// TIA Portal V20 export
// export: Created 2026-04-28T10:07:59.704243Z, ExportSetting WithDefaults, DisplayName Totally Integrated Automation Portal, DisplayVersion V20, DisplayName TIA Portal Openness, DisplayVersion V20, DisplayName TIA Portal Version Control Interface, DisplayVersion V20, DisplayName SINAMICS Startdrive Advanced, DisplayVersion V20, DisplayName SINAMICS Startdrive G130, G150, S120, S150, SINAMICS MV, G220, S200, S210, DisplayVersion V20, DisplayName SINAMICS Startdrive G110M, G120, G120C, G120D, G120P, G115D, DisplayVersion V20, DisplayName STEP 7 Professional, DisplayVersion V20, DisplayName STEP 7 Safety, DisplayVersion V20, DisplayName WinCC Basic/Comfort/Advanced, DisplayVersion V20, DisplayName WinCC Unified, DisplayVersion V20
TYPE "Daten_SPT_60"
// stored: IsFailsafeCompliant false
   STRUCT
      xSlPu : Bool := false;   // Selection Slip Pump
      txt_cSlPu_1_2 : DInt := 0;   // Selection Slip Pump 1 or 2
      xSlPuSoll : Bool := false;   // Selection Slip Pump Set Value
      xSlPuIst : Bool := false;   // Selection Slip Pump Actual Value
      txt_rSlPu : DInt := 0;   // Set value Slip pump
      RangeSlPu : DInt := 0;   // Range Slip pump
      iTakt_1_SlPu : DInt := 0;   // Interval for recording the measured values
      iAnzWerte_1_SlP : DInt := 0;   // Number of measured values
      xs1PuIst_Mod : Bool := false;   // Selection 0-20mA = 0 ; 0-10V = 1
      xSlPuSoll2 : Bool := false;   // Selection Slip Pump 2 Set Value
      xSlPuIst2 : Bool := false;   // Selection Slip Pump 2 Actual Value
      txt_rSlPu2 : DInt := 0;   // Set value Slip pump 2
      RangeSlPu2 : DInt := 0;   // Range Slip pump 2
      iTakt_2_SlPu : DInt := 0;   // Interval for recording the measured values
      iAnzWerte_2_SlP : DInt := 0;   // Number of measured values
      xSlip : Bool := false;   // Selection Slip
      xPrSlContr : Bool := false;   // Selection Slip pressure control
      txt_PrSlControll : DInt := 0;   // Slip pressure (control)
      txt_PrSlToleranze : DInt := 0;   // Slip pressure (tolerance)
      txt_iPrSlTime : Time := T#0MS;   // Slip pressure Delay time
      xPrSl : Bool := false;   // Selection Slip pressure
      txt_rPrSlMa : DInt := 0;   // Slip pressure Max
      txt_max_rPrSlMa : DInt := 0;   // Slip pressure Input Limit
      RangeSlPr : DInt := 0;   // Range Slip pressure
      iTakt_PrSl : DInt := 0;   // Interval for recording the measured values
      iAnzWerte_PrSl : DInt := 0;   // Number of measured values
      xPrSl2 : Bool := false;   // Selection Slip pressure 2
      txt_rPrSlMa2 : DInt := 0;   // Slip pressure 2 Max
      txt_max_rPrSlMa2 : DInt := 0;   // Slip pressure 2 Input Limit
      RangeSlPr2 : DInt := 0;   // Range Slip pressure 2
      iTakt_PrSl2 : DInt := 0;   // Interval for recording the measured values
      iAnzWerte_PrSl2 : DInt := 0;   // Number of measured values
      rDiffSl1Sl2_Set : DInt := 0;   // Difference value of slip pressure 1 and 2
      xFlRa : Bool := false;   // Selection Mass flow
      txt_rFlRaMa : DInt := 0;   // Mass flow Max.
      txt_max_rFlRaMa : DInt := 0;   // Mass flow Input Limit
      RangeFlRa : DInt := 0;   // Range Mass flow
      iTakt_FlRa : DInt := 0;   // Interval for recording the measured values
      iAnzWerte_FlRa : DInt := 0;   // Number of measured values
      xMemBreak : Bool := false;   // Selection Membrane break
      xAir : Bool := false;   // Selection Air
      xPrAi : Bool := false;   // Selection Pressure atomizing air
      RangePrAi : DInt := 0;   // Range Pressure atomizing air
      iTakt_PrAi : DInt := 0;   // Interval for recording the measured values
      iAnzWerte_PrAi : DInt := 0;   // Number of measured values
      xCoAi : Bool := false;   // Selection Air flow nozzle
      txt_rCoAiMi : DInt := 0;   // Air flow nozzle Max.
      txt_max_rCoAiMi : DInt := 0;   // Air flow nozzle Input Limit
      RangeCoAi : DInt := 0;   // Range Air flow nozzle
      iTakt_CoAi : DInt := 0;   // Interval for recording the measured values
      iAnzWerte_CoAi : DInt := 0;   // Number of measured values
      xSlSupp : Bool := false;   // Selection Slip feed
      xTankLevel : Bool := false;   // Selection Tank Level
      txt_iTankLevOver : DInt := 0;   // Tank Level Overflow
      txt_iTankLevMax : DInt := 0;   // Tank Level Max.
      txt_iTankLevMin : DInt := 0;   // Tank Level Min.
      iRangeTankLevel : DInt := 0;   // Range Tank Level
      iTakt_TankLevel : DInt := 0;   // Interval for recording the measured values
      iAnW_TankLevel : DInt := 0;   // Number of measured values
      xAgit_1 : Bool := false;   // Selection Agitator 1
      xAgitSoll_1 : Bool := false;   // Selection Agitator 1 Set Value
      xAgitIst_1 : Bool := false;   // Selection Agitator 1 Actual Value
      xAgitSpCon_1 : Bool := false;   // Selection Agitator 1 Speed ​​manual
      iRangeAgit_1 : DInt := 0;   // Range Agitator 1
      iAgitSoll_1 : DInt := 0;   // Set Value Agitator 1
      iTakt_Agit_1 : DInt := 0;   // Interval for recording the measured values
      iAnW_Agit_1 : DInt := 0;   // Number of measured values
      xScAgit_1 : Bool := false;   // Selection Scale agitator 1
      xScAgitSoll_1 : Bool := false;   // Selection Scale agitator 1 Set Value
      xScAgitIst_1 : Bool := false;   // Selection Scale agitator 1 Actual Value
      iRangeScAgit_1 : DInt := 0;   // Range Scale agitator 1
      iScAgitSoll_1 : DInt := 0;   // Set Value Scale agitator 1
      iScAgitMax_1 : DInt := 0;   // Scale agitator 1 Max
      iScAgitMin_1 : DInt := 0;   // Scale agitator 1 Min.
      iScAgitOver_1 : DInt := 0;   // Scale agitator 1 Over
      iTakt_ScAgit_1 : DInt := 0;   // Interval for recording the measured values
      iAnW_ScAgit_1 : DInt := 0;   // Number of measured values
      xAgit_2 : Bool := false;   // Selection Agitator 2
      xAgitSoll_2 : Bool := false;   // Selection Agitator 2 Set Value
      xAgitIst_2 : Bool := false;   // Selection Agitator 2 Actual Value
      xAgitSpCon_2 : Bool := false;   // Selection Agitator 2 Speed ​​manual
      iRangeAgit_2 : DInt := 0;   // Range Agitator 2
      iAgitSoll_2 : DInt := 0;   // Set Value Agitator 2
      iTakt_Agit_2 : DInt := 0;   // Interval for recording the measured values
      iAnW_Agit_2 : DInt := 0;   // Number of measured values
      xScAgit_2 : Bool := false;   // Selection Scale agitator 2
      xScAgitSoll_2 : Bool := false;   // Selection Scale agitator 2 Set Value
      xScAgitIst_2 : Bool := false;   // Selection Scale agitator 2 Actual Value
      iRangeScAgit_2 : DInt := 0;   // Range Scale agitator 2
      iScAgitSoll_2 : DInt := 0;   // Set Value Scale agitator 2
      iScAgitMax_2 : DInt := 0;   // Scale agitator 2 Max
      iScAgitMin_2 : DInt := 0;   // Scale agitator 2 Min.
      iScAgitOver_2 : DInt := 0;   // Scale agitator 2 Over
      iTakt_ScAgit_2 : DInt := 0;   // Interval for recording the measured values
      iAnW_ScAgit_2 : DInt := 0;   // Number of measured values
      xAgit_3 : Bool := false;   // Selection Agitator 3
      xAgitSoll_3 : Bool := false;   // Selection Agitator 3 Set Value
      xAgitIst_3 : Bool := false;   // Selection Agitator 3 Actual Value
      xAgitSpCon_3 : Bool := false;   // Selection Agitator 3 Speed ​​manual
      iRangeAgit_3 : DInt := 0;   // Range Agitator 3
      iAgitSoll_3 : DInt := 0;   // Set Value Agitator 3
      iTakt_Agit_3 : DInt := 0;   // Interval for recording the measured values
      iAnW_Agit_3 : DInt := 0;   // Number of measured values
      xScAgit_3 : Bool := false;   // Selection Scale agitator 3
      xScAgitSoll_3 : Bool := false;   // Selection Scale agitator 3 Set Value
      xScAgitIst_3 : Bool := false;   // Selection Scale agitator 3 Actual Value
      iRangeScAgit_3 : DInt := 0;   // Range Scale agitator 3
      iScAgitSoll_3 : DInt := 0;   // Set Value Scale agitator 3
      iScAgitMax_3 : DInt := 0;   // Scale agitator 3 Max
      iScAgitMin_3 : DInt := 0;   // Scale agitator 3 Min.
      iScAgitOver_3 : DInt := 0;   // Scale agitator 3 Over
      iTakt_ScAgit_3 : DInt := 0;   // Interval for recording the measured values
      iAnW_ScAgit_3 : DInt := 0;   // Number of measured values
      xAgit_4 : Bool := false;   // Selection Agitator 4
      xAgitSoll_4 : Bool := false;   // Selection Agitator 4 Set Value
      xAgitIst_4 : Bool := false;   // Selection Agitator 4 Actual Value
      xAgitSpCon_4 : Bool := false;   // Selection Agitator 4 Speed ​​manual
      iRangeAgit_4 : DInt := 0;   // Range Agitator 4
      iAgitSoll_4 : DInt := 0;   // Set Value Agitator 4
      iTakt_Agit_4 : DInt := 0;   // Interval for recording the measured values
      iAnW_Agit_4 : DInt := 0;   // Number of measured values
      xScAgit_4 : Bool := false;   // Selection Scale agitator 4
      xScAgitSoll_4 : Bool := false;   // Selection Scale agitator 4 Set Value
      xScAgitIst_4 : Bool := false;   // Selection Scale agitator 4 Actual Value
      iRangeScAgit_4 : DInt := 0;   // Range Scale agitator 4
      iScAgitSoll_4 : DInt := 0;   // Set Value Scale agitator 4
      iScAgitMax_4 : DInt := 0;   // Scale agitator 4 Max
      iScAgitMin_4 : DInt := 0;   // Scale agitator 4 Min.
      iScAgitOver_4 : DInt := 0;   // Scale agitator 4 Over
      iTakt_ScAgit_4 : DInt := 0;   // Interval for recording the measured values
      iAnW_ScAgit_4 : DInt := 0;   // Number of measured values
      xOelTemp : Bool := false;   // Selection Oil temperature slip pump
      iRangeOelTemp : DInt := 0;   // Range Oil temperature slip pump
      iTakt_OelTemp : DInt := 0;   // Interval for recording the measured values
      iAnW_OelTemp : DInt := 0;   // Number of measured values
      iSpOelTemp_1 : DInt := 0;   // Switching point 1 oil temperature slip pump
      iSpOelTemp_2 : DInt := 0;   // Switching point 2 oil temperature slip pump
      xNoS1SuppValve : Bool := false;   // Selection with/without switching valve
      t_iSlSuppContr : Time := T#0MS;   // Monitoring time switching water/slip
      txt_rSlPuWater : DInt := 0;   // Slip pressure at Di water
      t_iSuppSl_Wa : Time := T#0MS;   // Delay time switching water/slip
      xViscosity1 : Bool := false;   // Selection Viscosity 1 measurement
      RangeViscosity1 : DInt := 0;   // Range Viscosity 1 measurement
      iTakt_Viscosity1 : DInt := 0;   // Interval for recording the measured values
      iAnzWerte_Viscosity1 : DInt := 0;   // Number of measured values
      xViscosity2 : Bool := false;   // Selection Viscosity 2 measurement
      RangeViscosity2 : DInt := 0;   // Range Viscosity 2 measurement
      iTakt_Viscosity2 : DInt := 0;   // Interval for recording the measured values
      iAnzWerte_Viscosity2 : DInt := 0;   // Number of measured values
      RangeFlRaOffset : DInt := 0;   // Range Flowmeter offset input signal
      xSlPuControl : Bool := false;   // Selection Slip pump control
      RangeSlPuControl : DInt := 0;   // Range Slip pump control
      iTakt_SlPuControl : DInt := 0;   // Interval for recording the measured values
      iAnzWerte_SlPuControl : DInt := 0;   // Number of measured values
      rXp_PrCtrl : DInt := 0;   // Control P-Value Slip pump control
      rTi_PrCtrl : DInt := 0;   // Control I-Value Slip pump control
      rTd2_PrCtrl : DInt := 0;   // Control D-Value Slip pump control
      xSlPuControlHW : Bool := false;   // Selection Slip pump control Hardware
      xSlCtrlExt : Bool := false;   // Slip Pumpe External Start/Stop
      xSlPu_Set_4_20mA : Bool := false;   // SetValue for the pump 4 - 20 mA 1 = Yes; 0 = No
      xMemBreak_2 : Bool := false;   // Selection Membrane break 2
      xPrSlCtrl_Intervall : Bool := false;   // Selection Slip pressure monitoring at defined intervals
      txt_rPrSlCtrl_Up : DInt := 0;   // Slip pressure monitoring at defined intervals Up
      txt_rPrSlCtrl_Down : DInt := 0;   // Slip pressure monitoring at defined intervals Below
      xPrFLRa_Intervall : Bool := false;   // Selection Slip quantity monitoring at defined intervals
      txt_PrFLRaCtrl_Up : DInt := 0;   // Slip quantity monitoring at defined intervals Up
      txt_PrFLRaCtrl_Down : DInt := 0;   // Slip quantity monitoring at defined intervals Below
      xSlTe : Bool;   // Selection Slip Temperature
      txt_rSlTeMa : DInt;   // Slip Temperature Max.
      xZSS_Option : Bool;   // Selection Atomizer disc
      Range_ZSS_Istwert : DInt;   // Range Atomizer disc Act. Value
      xMAUF_Option : Bool;   // Selection Mass preparation
      RangeSlPr_D20 : DInt := 0;   // Range Slip pressure
      txt_rPrSlMa_D20 : DInt := 0;   // Slip pressure Max
      txt_max_rPrSlMa_D20 : DInt := 0;   // Slip pressure Input Limit
      txt_rFlRaMa_D20 : DInt := 0;   // Mass flow Max.
      txt_max_rFlRaMa_D20 : DInt := 0;   // Mass flow Input Limit
      RangeFlRa_D20 : DInt := 0;   // Range Mass flow
   END_STRUCT;
END_TYPE
